(*
SPDX-FileCopyrightText: © 2026 Oleksandr Tiutyk <trofimich@gmail.com>
SPDX-License-Identifier: MIT
License: https://opensource.org/license/mit
*)

(*!
<summary>Provides automation components with indexed access to their related objects.</summary>
<description>
Indexed Try lookups borrow interfaces and contain exceptions. Fatal allocation observations return null
without clearing the latch.
A state transition during output processing skips remaining outputs and the after-output hook.
Completed writes remain effective. A pass started in STOPPED proceeds while the branch stays in that state.
Parent is mandatory and borrowed for the component lifetime.
</description>
*)

FUNCTION_BLOCK ABSTRACT CompositeAutomationComponent
VAR_GENERIC CONSTANT
	{attribute 'hide'} 
    _ChildCount : TOF_Core.INT_LENGTH := 0;
END_VAR
EXTENDS BranchAutomationComponent IMPLEMENTS ICompositeAutomationComponent
VAR
	{attribute 'hide'} 
	_Parent : IParentAutomationComponent;
END_VAR

METHOD FINAL BubbleEvent
VAR_INPUT
	event : TOF_Core.IEvent;
END_VAR
VAR
	stopPropagation : BOOL;
	
	parentAsBubbleEventDispatcher : TOF_Core.IBubbleEventDispatcher;
END_VAR
OnEventReceived(event := event, stopPropagation => stopPropagation);

IF stopPropagation THEN
	RETURN;
END_IF

IF __QUERYINTERFACE(Parent, parentAsBubbleEventDispatcher) THEN
	parentAsBubbleEventDispatcher.BubbleEvent(event := event);
END_IF
END_METHOD

{attribute 'monitoring' := 'call'}
PROPERTY FINAL ChildCount : TOF_Core.INT_LENGTH
GET
ChildCount := _ChildCount;
END_GET
END_PROPERTY

{attribute 'monitoring' := 'call'}
PROPERTY ABSTRACT Children : REFERENCE TO ARRAY [0.._ChildCount - 1] OF IChildAutomationComponent
GET
END_GET
END_PROPERTY

METHOD FB_init : BOOL
VAR_INPUT
	bInitRetains : BOOL; // TRUE: the retain variables are initialized (reset warm / reset cold)
	bInCopyCode : BOOL;  // TRUE: the instance will be copied to the copy code afterward (online change)
	name : WSTRING;
	parent : IParentAutomationComponent;
END_VAR
_Parent := parent;
END_METHOD

(*!
<summary>Borrows the constructor-bound parent for the composite lifetime.</summary>
<description>
The parent is mandatory for initialization and must remain live. Ownership is not transferred.
</description>
*)
{attribute 'monitoring' := 'call'}
PROPERTY FINAL Parent : IParentAutomationComponent
GET
Parent := _Parent;
END_GET
END_PROPERTY

(*!
<summary>Processes enabled input children in slot order.</summary>
<description>
While the branch remains enabled, a transition to STOPPED continues the input pass through the remaining
enabled input children and the after-input hook. Input callbacks must support execution in STOPPED.
</description>
*)
METHOD FINAL ProcessInput
VAR
	exceptionCode : __SYSTEM.ExceptionCode;
	exception : TOF_Core.IException;	
	exceptionReaction : TOF_Core.EXCEPTION_REACTION;
	
	childCriticalErrorReaction : CHILD_CRITICAL_ERROR_REACTION;
	
	i : INT;
		
	child : IChildAutomationComponent;	

	inputDevice : IInputLeafAutomationComponent;
END_VAR
__TRY
	OnBeforeChildrenProcessInput();
__CATCH(exceptionCode)		
	exception := TOF_Core.ExceptionManager.GetLastException(
		exceptionCode := exceptionCode,
		catchPointNamespaceName := NamespaceName,
		catchPointPOUName := __POUNAME(),
		catchPointPosition := __POSITION()
	);
					
	exceptionReaction := OnHandleException(exception := exception, failedMethodName := 'OnBeforeChildrenProcessInput');

	ProcessException(
		exception := exception,
		exceptionReaction := exceptionReaction,
		exceptionSourceHint := "OnBeforeChildrenProcessInput error"
	);
__ENDTRY

FOR i := 0 TO _ChildCount - 1 DO
	child := TryGetChildByIndex(index := i);

	IF child = 0 OR_ELSE NOT child.Enabled OR_ELSE NOT __QUERYINTERFACE(child, inputDevice) THEN
		CONTINUE;
	END_IF
	
	inputDevice.ProcessInput();

	IF inputDevice.HasError AND_THEN inputDevice.Error.Severity = TOF_Core.ERROR_SEVERITY.CRITICAL THEN
		childCriticalErrorReaction := HandleChildCriticalError(childWithError := inputDevice);
		
		ProcessChildError(
			childError := inputDevice.Error,
			childErrorReaction := childCriticalErrorReaction,
			childErrorSourceHint := TOF_Core.WideStrings.Concat255(
				"Child[",
				TO_WSTRING(i),
				"](",
				inputDevice.Name,
				").ProcessInput error"
			)
		);
	END_IF		
END_FOR

__TRY
	OnAfterChildrenProcessInput();
__CATCH(exceptionCode)		
	exception := TOF_Core.ExceptionManager.GetLastException(
		exceptionCode := exceptionCode,
		catchPointNamespaceName := NamespaceName,
		catchPointPOUName := __POUNAME(),
		catchPointPosition := __POSITION()
	);
					
	exceptionReaction := OnHandleException(exception := exception, failedMethodName := 'OnAfterChildrenProcessInput');

	ProcessException(
		exception := exception,
		exceptionReaction := exceptionReaction,
		exceptionSourceHint := "OnAfterChildrenProcessInput error"
	);
__ENDTRY
END_METHOD

(*!
<summary>Processes enabled output children in slot order.</summary>
<description>
A state transition during output processing skips remaining outputs and the after-output hook.
Completed writes remain effective. A pass started in STOPPED proceeds while the branch stays in that state.
</description>
*)
METHOD FINAL ProcessOutput
VAR
	entryRevision : UDINT;
	exceptionCode : __SYSTEM.ExceptionCode;
	exception : TOF_Core.IException;	
	exceptionReaction : TOF_Core.EXCEPTION_REACTION;
	
	childCriticalErrorReaction : CHILD_CRITICAL_ERROR_REACTION;
	
	i : INT;
		
	child : IChildAutomationComponent;	

	outputDevice : IOutputLeafAutomationComponent;
END_VAR
entryRevision := _OperationalStateRevision;

__TRY
	OnBeforeChildrenProcessOutput();
__CATCH(exceptionCode)		
	exception := TOF_Core.ExceptionManager.GetLastException(
		exceptionCode := exceptionCode,
		catchPointNamespaceName := NamespaceName,
		catchPointPOUName := __POUNAME(),
		catchPointPosition := __POSITION()
	);
					
	exceptionReaction := OnHandleException(exception := exception, failedMethodName := 'OnBeforeChildrenProcessOutput');

	ProcessException(
		exception := exception,
		exceptionReaction := exceptionReaction,
		exceptionSourceHint := "OnBeforeChildrenProcessOutput error"
	);
__ENDTRY

FOR i := 0 TO _ChildCount - 1 DO
	IF _OperationalStateRevision <> entryRevision THEN
		RETURN;
	END_IF

	child := TryGetChildByIndex(index := i);

	IF child = 0 OR_ELSE NOT child.Enabled OR_ELSE NOT __QUERYINTERFACE(child, outputDevice) THEN
		CONTINUE;
	END_IF
	
	IF _OperationalStateRevision <> entryRevision THEN
		RETURN;
	END_IF

	outputDevice.ProcessOutput();
	
	IF outputDevice.HasError AND_THEN outputDevice.Error.Severity = TOF_Core.ERROR_SEVERITY.CRITICAL THEN
		childCriticalErrorReaction := HandleChildCriticalError(childWithError := outputDevice);
		
		ProcessChildError(
			childError := outputDevice.Error,
			childErrorReaction := childCriticalErrorReaction,
			childErrorSourceHint := TOF_Core.WideStrings.Concat255(
				"Child[",
				TO_WSTRING(i),
				"](",
				outputDevice.Name,
				").ProcessOutput error"
			)
		);
	END_IF
END_FOR

IF _OperationalStateRevision <> entryRevision THEN
	RETURN;
END_IF

__TRY
	OnAfterChildrenProcessOutput();
__CATCH(exceptionCode)		
	exception := TOF_Core.ExceptionManager.GetLastException(
		exceptionCode := exceptionCode,
		catchPointNamespaceName := NamespaceName,
		catchPointPOUName := __POUNAME(),
		catchPointPosition := __POSITION()
	);
					
	exceptionReaction := OnHandleException(exception := exception, failedMethodName := 'OnAfterChildrenProcessOutput');

	ProcessException(
		exception := exception,
		exceptionReaction := exceptionReaction,
		exceptionSourceHint := "OnAfterChildrenProcessOutput error"
	);
__ENDTRY
END_METHOD

(*!
<summary>Returns a borrowed child by its zero-based index.</summary>
<description>
Returns null when the entry is unavailable, the index is out of range or a nested call raises an exception.
Fatal allocation observations before or after the storage getter return null and preserve the latch for
the outer task boundary. Does not transfer ownership or extend lifetime. Getter exceptions are contained.
</description>
*)
METHOD FINAL TryGetChildByIndex : IChildAutomationComponent
VAR_INPUT
	index : TOF_Core.INT_INDEX;
END_VAR
VAR
	childStorage : REFERENCE TO ARRAY [0.._ChildCount - 1] OF IChildAutomationComponent;
END_VAR
__TRY
	IF TOF_Core.DynamicMemoryManager.HasAllocationFailed OR_ELSE index < 0 OR_ELSE index >= _ChildCount THEN
		RETURN;
	END_IF

	childStorage REF= Children;

	IF NOT TOF_Core.DynamicMemoryManager.HasAllocationFailed AND_THEN __ISVALIDREF(childStorage) THEN
		TryGetChildByIndex := childStorage[index];
	END_IF
__CATCH
	TryGetChildByIndex := 0;
__ENDTRY

IF TOF_Core.DynamicMemoryManager.HasAllocationFailed THEN
	TryGetChildByIndex := 0;
END_IF
END_METHOD

METHOD PROTECTED FINAL Validate
VAR
END_VAR
IF _Parent = 0 THEN
	TOF_Core.Exceptions.ThrowDataMemberNotSpecified(
		sourceNamespaceName := NamespaceName,
		sourceClassName := ClassName,
		sourcePOUName := __POUNAME(),
		sourcePosition := __POSITION(),
		dataMemberName := 'Parent'
	);						
END_IF

IF ChildCount > 0 AND_THEN NOT __ISVALIDREF(Children) THEN
	TOF_Core.Exceptions.ThrowDataMemberNotSpecified(
		sourceNamespaceName := NamespaceName,
		sourceClassName := ClassName,
		sourcePOUName := __POUNAME(),
		sourcePosition := __POSITION(),
		dataMemberName := 'Children'
	);
END_IF
END_METHOD

END_FUNCTION_BLOCK

(* stored: Version 1.1.0.1
   POU CompositeAutomationComponent: Id {25bfda0d-9225-4be2-8314-f8314e830df8}, SpecialFunc None
   Folder Overriden methods: Id {8e7fddf3-79b8-4a8a-9258-2efb57fe9a7d}
   Method BubbleEvent: Id {ec63c85f-f731-4851-bd8e-f85a62e07837}
   Property ChildCount: Id {eab6dfe5-2f53-4cc8-87ce-0fc821a75f9c}
   Get Get: Id {46ef8b88-c91b-4061-8848-8d8aa1c34fff}
   Property Children: Id {5eb8cc14-af21-41a6-964e-854d2107c6da}
   Get Get: Id {92c9163e-e171-4a3b-8e8e-5251e6af78eb}
   Method FB_init: Id {515605cc-0879-42b7-b0de-34f0ad85bef8}
   Property Parent: Id {8abf624b-c9ed-4996-8788-b464b8e15520}
   Get Get: Id {872e7375-00a6-46e3-b1e4-754a1ea8aef4}
   Method ProcessInput: Id {169f608c-73af-42d0-b266-fd32baea3032}
   Method ProcessOutput: Id {d8822de7-f12d-43fe-bdcd-3812e5246f80}
   Method TryGetChildByIndex: Id {d6468cc2-d65d-413d-b788-a326d0027f11}
   Method Validate: Id {cbb4acd1-d175-4a92-bf2b-4e4a64c68356} *)
